FUNCTION_BLOCK FB_VSIStorageSystem EXTENDS FB_SystemContinous
VAR_INPUT
	bLoadingAutomatic : BOOL; //variable to determine if storage is in loading mode
	aTelegramm_WMZ305 : ARRAY[1..cMBUS_MaxTelegrams] OF ST_MBus_Data2;
END_VAR
VAR_OUTPUT
	localState : ST_VSIStorageState;
END_VAR
VAR
	{attribute 'OPC.UA.DA' := '1'}
	localSetParameters : ST_VSIStorageSetParameters;
	
	//default parameters
	localDefaultParameters : ST_VSIStorageSystemDefaultParameters;	

	//storage
	VSIStorage : FB_VSIStorage;
	
	//pumps
	
	stPU305DefaultParameters : ST_PumpGrundfosMagna3DefaultParameters := (bExternalTemperatureSensor := FALSE);
	PU305 : FB_PumpGrundfosMagna3 := (ST_DefaultParameters := stPU305DefaultParameters);; //Magna 3 pump (loading pump)
	PU306 : FB_PumpGrundfosMagna3 := (ST_DefaultParameters := stPU305DefaultParameters);; //Magna 3 pump (unloading pump)

	//valves
	stSV305DefaultParameters : ST_MixingValveDefaultParameters := (tTaskCycleTime := GlobalVariables.tCtrlCycleTime_MAIN, tCtrlCycleTime := GlobalVariables.tCtrlCycleTime_MAIN);
	stSV306DefaultParameters : ST_MixingValveDefaultParameters := (tTaskCycleTime := GlobalVariables.tCtrlCycleTime_MAIN, tCtrlCycleTime := GlobalVariables.tCtrlCycleTime_MAIN);
	stSV307DefaultParameters : ST_MixingValveDefaultParameters := (tTaskCycleTime := GlobalVariables.tCtrlCycleTime_MAIN, tCtrlCycleTime := GlobalVariables.tCtrlCycleTime_MAIN);
	
	SV305 : FB_MixingValve := (ST_DefaultParameters := stSV305DefaultParameters); //discrete inlet valve, valve motor needs continous signal but operates only between extreme positions
	SV306 : FB_MixingValve := (ST_DefaultParameters := stSV306DefaultParameters); //discrete outlet valve	, valve motor needs continous signal but operates only between extreme positions
	SV307 : FB_MixingValve := (ST_DefaultParameters := stSV307DefaultParameters); //discrete outlet valve	, valve motor needs continous signal but operates only between extreme positions
	
	//sensors
	WMZ305 : FB_MollineC3HeatCounter;
	
	//internal variables
	bSetStatusOn_PU305 : BOOL;
	bSetStatusOn_PU306 : BOOL;
	bSetStatusOn_SV305 : BOOL;
	fSetPoint_SV305 : REAL;
	bSetStatusOn_SV306 : BOOL;
	fSetPoint_SV306 : REAL;
	bSetStatusOn_SV307 : BOOL;
	fSetPoint_SV307 : REAL;
	bLoading : BOOL;
	
	//triggers
	SwitchToLoading : R_TRIG;
	SwitchToUnloading : F_TRIG;
	bFinishedSwitchMode : BOOL := TRUE;
END_VAR

//storage
VSIStorage(localState => localState);

SelectLoadingMode();
SwitchToLoading(CLK := bLoading);
SwitchToUnloading(CLK := bLoading);

//MAIN must be called before SwitchMode to prevent pump signal chattering (signal is written after SwitchMode function), SwitchMode may only be called if system is on
MAIN();

//disrupt calling SystemFlowControl via MAIN() when mode is switched and call SwitchMode()
IF ((SwitchToLoading.Q OR SwitchToUnloading.Q) OR NOT bFinishedSwitchMode) AND bSetStatusOn THEN
	SwitchMode(bSwitchToLoading := bLoading,
		bFinishedSwitchMode => bFinishedSwitchMode);
END_IF;

//pumps
PU305.GetState_Profibus();
PU305(bSetStatusOnAutomatic := bSetStatusOn_PU305,
	fSetPointAutomatic := fSetPoint,
	bAlgorithmPermission := bAlgorithmPermission,
	nControlModeAutomatic := 0);
PU305.SetState_Profibus();

PU306.GetState_Profibus();
PU306(bSetStatusOnAutomatic := bSetStatusOn_PU306,
	fSetPointAutomatic := fSetPoint,
	bAlgorithmPermission := bAlgorithmPermission,
	nControlModeAutomatic := 0);
PU306.SetState_Profibus();

//valves
SV305.GetState_AI();
SV305(bSetStatusOnAutomatic := bSetStatusOn_SV305,
	fSetPointAutomatic := fSetPoint_SV305,
	bAlgorithmPermission := bAlgorithmPermission,
	nControlModeAutomatic := 0);
SV305.SetState_AO();

SV306.GetState_AI();
SV306(bSetStatusOnAutomatic := bSetStatusOn_SV306,
	fSetPointAutomatic := fSetPoint_SV306,
	bAlgorithmPermission := bAlgorithmPermission,
	nControlModeAutomatic := 0);
SV306.SetState_AO();

SV307.GetState_AI();
SV307(bSetStatusOnAutomatic := bSetStatusOn_SV307,
	fSetPointAutomatic := 100,
	bAlgorithmPermission := bAlgorithmPermission,
	nControlModeAutomatic := 0);
SV307.SetState_AO();

//insert heat counter telegramm from other task
WMZ305(aHeatCounterTelegramm := aTelegramm_WMZ305);

METHOD PROTECTED  CheckError : BOOL
VAR_INPUT
END_VAR
VAR_OUTPUT
	bError : BOOL;
END_VAR
VAR
	bError_PUx05 : BOOL;
END_VAR
//check for pump error
bError_PUx05 := PU305.bError OR PU306.bError;
END_METHOD

METHOD PROTECTED  Operational : BOOL
VAR_INPUT
END_VAR
VAR_OUTPUT
	bSwitchToWorking : BOOL := FALSE;
END_VAR
IF PU305.bStatusOn OR PU306.bStatusOn THEN
	bSwitchToWorking := TRUE;
END_IF
END_METHOD

METHOD PROTECTED  RampDown : BOOL
VAR_INPUT
END_VAR
VAR_OUTPUT
	bRampDownFinished : BOOL := FALSE;
END_VAR
bSetStatusOn_PU305 := FALSE;
bSetStatusOn_PU306 := FALSE;

IF NOT PU305.bStatusOn AND NOT PU306.bStatusOn THEN
	bSetStatusOn_SV305 := FALSE;
	bSetStatusOn_SV306 := FALSE;
	bSetStatusOn_SV307 := FALSE;
	IF SV305.fOperatingPoint<20 AND SV306.fOperatingPoint<20 AND SV307.fOperatingPoint<20 THEN
		bRampDownFinished := TRUE;
	END_IF
END_IF
END_METHOD

METHOD PROTECTED  RampUp : BOOL
VAR_INPUT
END_VAR
VAR_OUTPUT
	bRampUpFinished : BOOL := FALSE;
END_VAR
bSetStatusOn_SV305 := TRUE;
bSetStatusOn_SV306 := TRUE;
bSetStatusOn_SV307 := TRUE;

IF bLoading THEN
	fSetPoint_SV305 := 100;
	fSetPoint_SV306 := 0;
	IF SV305.fOperatingPoint>80 AND SV306.fOperatingPoint<20 AND SV307.fOperatingPoint>80 THEN
		bSetStatusOn_PU305 := TRUE;	
		bSetStatusOn_PU306 := FALSE;	
		bRampUpFinished := TRUE;	
	END_IF
ELSE
	fSetPoint_SV305 := 0;
	fSetPoint_SV306 := 100;
	IF SV305.fOperatingPoint<20 AND SV306.fOperatingPoint>80 AND SV307.fOperatingPoint>80 THEN
		bSetStatusOn_PU305 := FALSE;	
		bSetStatusOn_PU306 := TRUE;		
		bRampUpFinished := TRUE;
	END_IF
END_IF
END_METHOD

METHOD PRIVATE SelectLoadingMode : BOOL
VAR_INPUT
END_VAR
IF control.bManualModeActivated THEN
	bLoading := localSetParameters.bLoadingManual;
ELSIF control.bAlgorithmModeActivated AND bAlgorithmPermission THEN
	bLoading := localSetParameters.bLoadingAlgorithm;
ELSE
	bLoading := bLoadingAutomatic;
END_IF
END_METHOD

METHOD PROTECTED   SetSetPointLimits : BOOL
VAR_INPUT
END_VAR
aSetPointLimits[1] := localDefaultParameters.aSetPointLimitsTemperature[1];
aSetPointLimits[2] := localDefaultParameters.aSetPointLimitsTemperature[2];
END_METHOD

METHOD PROTECTED  SetState : BOOL
VAR_INPUT
END_VAR
VAR_OUTPUT
END_VAR
IF bLoading THEN
	fOperatingPoint := PU305.fOperatingPoint;
ELSE
	fOperatingPoint := PU306.fOperatingPoint;
END_IF
controlState.bStatusOn := bSetStatusOn;
setPointState.aSetPointLimits := aSetPointLimits;
setPointState.fSetPoint := fSetPoint;
setPointState.fOperatingPoint := fOperatingPoint;
setPointState.sSetPointUnit := 'percent';
setPointState.sOperatingPointUnit := 'percent';
END_METHOD

PROPERTY ST_DefaultParameters : REFERENCE TO ST_VSIStorageSystemDefaultParameters
SET
localDefaultParameters := ST_DefaultParameters;
END_SET
END_PROPERTY

METHOD PRIVATE SwitchMode : BOOL
VAR_INPUT
	bSwitchToLoading : BOOL; //if false switch to cooling
END_VAR
VAR_OUTPUT
	bFinishedSwitchMode : BOOL := FALSE;
END_VAR
VAR_INST
	bRampDownFinished : BOOL := FALSE;
END_VAR
//check system state
IF bRampDownFinished THEN
	IF bSwitchToLoading THEN
		fSetPoint_SV305 := 100;
		fSetPoint_SV306 := 0;
		IF SV305.fOperatingPoint>80 AND SV306.fOperatingPoint<20 THEN
			//reset instant variable and switch on pump
			bRampDownFinished := FALSE;			
			bFinishedSwitchMode := TRUE;
			bSetStatusOn_PU305 := TRUE;
		END_IF
		
	ELSE
		fSetPoint_SV305 := 0;
		fSetPoint_SV306 := 100;
		IF SV305.fOperatingPoint<20 AND SV306.fOperatingPoint>80 THEN
			//reset instant variable and switch on pump
			bRampDownFinished := FALSE;			
			bFinishedSwitchMode := TRUE;
			bSetStatusOn_PU306 := TRUE;
		END_IF
	END_IF
ELSE
	bSetStatusOn_PU305 := FALSE;
	bSetStatusOn_PU306 := FALSE;
	IF NOT PU305.bStatusOn AND NOT PU306.bStatusOn THEN
		bRampDownFinished := TRUE;
	END_IF
END_IF
END_METHOD

METHOD PROTECTED  Working : BOOL
VAR_INPUT
END_VAR
VAR_OUTPUT
	bSwitchToOperational : BOOL := FALSE;
END_VAR
//empty method
END_METHOD

END_FUNCTION_BLOCK

(* stored: Version 1.1.0.1, ProductVersion 3.1.4024.10
   POU FB_VSIStorageSystem: Id {382610c2-8efd-46b8-a6e8-c6c7263961ee}, SpecialFunc None
   Method CheckError: Id {e6500ceb-116e-45d5-85e5-f2a65c10cf67}
   Method Operational: Id {2b4ab98b-64cb-4298-bf01-c47a40f2848c}
   Method RampDown: Id {efc28074-0dab-4054-8444-a8e746ef0234}
   Method RampUp: Id {edbe4b00-58dc-45ef-b254-23ba45e5f41a}
   Method SelectLoadingMode: Id {874dd5e5-f3db-4d2a-986b-16df54211a39}
   Method SetSetPointLimits: Id {148b0422-ab65-4f9e-b546-627d400f8fe6}
   Method SetState: Id {8f1694a5-bd9d-4950-9191-74b047cf31a8}
   Property ST_DefaultParameters: Id {02e19c12-9389-4ce3-90cd-253fab447e26}
   Set Set: Id {c9f9f9ec-22e1-4654-8a73-f50ab5f29b54}
   Method SwitchMode: Id {61519c15-9009-463d-b564-433e6de7eb20}
   Method Working: Id {09007639-5a67-4258-af27-ae8424745105} *)
